Staubli VAL3: encodeShareReal.pgx

public program encodeShareReal(num& x_nStatus (dimensions=1), num& x_nOutputBuffer[] (dimensions=1), num& x_nBufferPos (dimensions=1), num x_nSharedReal (dimensions=1))
  local num l_nDWordBytes[4]
begin
  if x_nStatus<0
    return
  endIf
  x_nStatus=-1
  x_nStatus=toBinary(x_nSharedReal,1,"4.0l",l_nDWordBytes)
  if x_nStatus<0
    putln("Failed to encode shared real at index: "+toString("",x_nBufferPos)+", status: "+toString("",x_nStatus))
    return
  endIf
  call copyArray(x_nOutputBuffer,x_nBufferPos,l_nDWordBytes)

end
